{attribute 'qualified_only'}
{attribute 'strict'}
{attribute 'to_string'}
TYPE E_PodState :
(
	STATE_EMERGENCY		:= 0,
	STATE_BOOT 			:= 1,
    STATE_SYNC 			:= 2,
    STATE_IDLE 			:= 3,
    STATE_HV_ACTIVE		:= 4,
    STATE_DEMO			:= 5,
    STATE_LEVITATION	:= 6,
    STATE_MOVEMENT		:= 7,
    STATE_MAINTENANCE	:= 8
);
END_TYPE

(* stored: Version 1.1.0.1
   DUT E_PodState: Id {f59f6ad5-9f7c-4ee7-88c1-b58056b4c9fa} *)
